(* IEC 61131-3 sources: AXOpen/src/components.desoutter.tightening/app/SystemConstants, 2 files *)

(* ---- plc_line_IoAddresses.st ---- *)
CONFIGURATION IoAddresses
    VAR_GLOBAL

        // Module desoutter/Input_1_byte_1
        desoutter_Input_1_byte_1_Input AT %IB13 : desoutter_Input_1_byte_1_Input_Layout;

        // Module desoutter/Input_1_byte_2
        desoutter_Input_1_byte_2_Input AT %IB12 : desoutter_Input_1_byte_2_Input_Layout;

        // Module desoutter/Input_1_word_1
        desoutter_Input_1_word_1_Input AT %IB6 : desoutter_Input_1_word_1_Input_Layout;

        // Module desoutter/Input_1_word_2
        desoutter_Input_1_word_2_Input AT %IB0 : desoutter_Input_1_word_2_Input_Layout;

        // Module desoutter/Input_2_word_1
        desoutter_Input_2_word_1_Input AT %IB8 : desoutter_Input_2_word_1_Input_Layout;

        // Module desoutter/Input_2_word_2
        desoutter_Input_2_word_2_Input AT %IB2 : desoutter_Input_2_word_2_Input_Layout;

        // Module desoutter/Output_1_byte_1
        desoutter_Output_1_byte_1_Output AT %QB1 : desoutter_Output_1_byte_1_Output_Layout;

        // Module desoutter/Output_1_byte_2
        desoutter_Output_1_byte_2_Output AT %QB0 : desoutter_Output_1_byte_2_Output_Layout;
    END_VAR
END_CONFIGURATION

TYPE
    desoutter_Input_1_byte_1_Input_Layout : STRUCT
        Signals_0 AT %B0 : BYTE;
    END_STRUCT;
END_TYPE

TYPE
    desoutter_Input_1_byte_2_Input_Layout : STRUCT
        Signals_0 AT %B0 : BYTE;
    END_STRUCT;
END_TYPE

TYPE
    desoutter_Input_1_word_1_Input_Layout : STRUCT
        Signals_0 AT %B0 : WORD;
    END_STRUCT;
END_TYPE

TYPE
    desoutter_Input_1_word_2_Input_Layout : STRUCT
        Signals_0 AT %B0 : WORD;
    END_STRUCT;
END_TYPE

TYPE
    desoutter_Input_2_word_1_Input_Layout : STRUCT
        Signals_0 AT %B0 : DWORD;
    END_STRUCT;
END_TYPE

TYPE
    desoutter_Input_2_word_2_Input_Layout : STRUCT
        Signals_0 AT %B0 : DWORD;
    END_STRUCT;
END_TYPE

TYPE
    desoutter_Output_1_byte_1_Output_Layout : STRUCT
        Signals_0 AT %B0 : BYTE;
    END_STRUCT;
END_TYPE

TYPE
    desoutter_Output_1_byte_2_Output_Layout : STRUCT
        Signals_0 AT %B0 : BYTE;
    END_STRUCT;
END_TYPE

(* ---- plc_line_HwIdentifiers.st ---- *)
CONFIGURATION HardwareIDs
    VAR_GLOBAL CONSTANT
        desoutter_cvic_ii_HwID : UINT := UINT#258;
        desoutter_cvic_ii_Input_1_byte_1_Input_1_byte_HwID : UINT := UINT#269;
        desoutter_cvic_ii_Input_1_byte_2_Input_1_byte_HwID : UINT := UINT#268;
        desoutter_cvic_ii_Input_1_word_1_Input_1_word_HwID : UINT := UINT#266;
        desoutter_cvic_ii_Input_1_word_2_Input_1_word_HwID : UINT := UINT#264;
        desoutter_cvic_ii_Input_2_word_1_Input_2_word_HwID : UINT := UINT#267;
        desoutter_cvic_ii_Input_2_word_2_Input_2_word_HwID : UINT := UINT#265;
        desoutter_cvic_ii_Output_1_byte_1_Output_1_byte_HwID : UINT := UINT#263;
        desoutter_cvic_ii_Output_1_byte_2_Output_1_byte_HwID : UINT := UINT#262;
        desoutter_cvic_ii_Rack_HwID : UINT := UINT#260;
        desoutter_cvic_ii_desoutter_cvic_ii_HwID : UINT := UINT#261;
        desoutter_cvic_ii_desoutter_cvic_ii_Interface_HwID : UINT := UINT#257;
        desoutter_cvic_ii_desoutter_cvic_ii_Interface_Port_1_HwID : UINT := UINT#259;
        desoutter_cvic_ii_desoutter_cvic_ii_RT_HwID : UINT := UINT#270;
        plc_line_HwID : UINT := UINT#32;
        plc_line_Rail_0_HwID : UINT := UINT#271;
        plc_line_plc_line_HwID : UINT := UINT#48;
        plc_line_plc_line_CPU_display_1_HwID : UINT := UINT#54;
        plc_line_plc_line_Card_reader_writer_1_HwID : UINT := UINT#51;
        plc_line_plc_line_DP_interface_1_HwID : UINT := UINT#60;
        plc_line_plc_line_OPC_UA_1_HwID : UINT := UINT#117;
        plc_line_plc_line_PROFINET_interface_1_HwID : UINT := UINT#64;
        plc_line_plc_line_PROFINET_interface_1_Port_1_HwID : UINT := UINT#65;
        plc_line_plc_line_PROFINET_interface_1_Port_2_HwID : UINT := UINT#66;
        plc_line_plc_line_PROFINET_interface_2_HwID : UINT := UINT#72;
        plc_line_plc_line_PROFINET_interface_2_Port_3_HwID : UINT := UINT#73;
        plc_line_plc_line_Virtual_communication_interface_HwID : UINT := UINT#135;
        profinet_plc_line_HwID : UINT := UINT#256;

    END_VAR
END_CONFIGURATION
